// TIA Portal V20 export
VAR_GLOBAL   // PLC tag table "Robot_Efort"
   Mission_Command AT %QW524 : Int;   // Invio delle missioni a robot
   "X_Pick-Place_LOW" AT %QW526 : Int;
   "Y_Pick-Place_LOW" AT %QW530 : Int;
   "Z_Pick-Place_LOW" AT %QW534 : Int;
   "ZRot_Pick-Place_LOW" AT %QW538 : Int;
   "YRot_Pick-Place_LOW" AT %QW542 : Int;
   "XRot_Pick-Place_LOW" AT %QW546 : Int;
   Gripper_code AT %QW550 : Int;
   Gripper1_XDim_LOW AT %QW552 : Int;
   Gripper1_YDim_LOW AT %QW556 : Int;
   Gripper1_ZDim_LOW AT %QW560 : Int;
   Gripper1_ZRotDim_LOW AT %QW564 : Int;
   Gripper1_YRotDim_LOW AT %QW568 : Int;
   Gripper1_XRotDim_LOW AT %QW572 : Int;
   Gripper2_XDim_LOW AT %QW576 : Int;
   Gripper2_YDim_LOW AT %QW580 : Int;
   Gripper2_ZDim_LOW AT %QW584 : Int;
   Gripper2_ZRotDim_LOW AT %QW588 : Int;
   Gripper2_YRotDim_LOW AT %QW592 : Int;
   Gripper2_XRotDim_LOW AT %QW596 : Int;
   X_approach_LOW AT %QW600 : Int;
   Y_approach_LOW AT %QW604 : Int;
   Z_approach_LOW AT %QW608 : Int;
   ZRot_approach_LOW AT %QW612 : Int;
   YRot_approach_LOW AT %QW616 : Int;
   XRot_approach_LOW AT %QW620 : Int;
   ApproachType AT %QW624 : Int;   // 1 XX, 2 YY, 3 ZZ, 4 XZ, 5 ZX, 6 YZ, 7 ZY, 8 XY , 9 YX
   Unit_code AT %QW626 : Int;   // 1-4 warehouse, 11-14 Machines 1→4, 21-29 grippers positions 1→9 on shelf
   Object_Type AT %QW628 : Int;   // 1 Part, 2 vice, 3 pallet, 4 gripper
   Gripper_Side AT %QW632 : Int;   // 1 RAW, 2 fFINISHED
   cmd_Status_PalletLocked AT %Q503.0 : Bool;   // segnale di pallet bloccato
   cmd_Status_PalletUnlocked AT %Q503.1 : Bool;   // segnale di pallet sbloccato
   cmd_status_Vice_locked AT %Q503.2 : Bool;   // segnale di morsa chiusa
   cmd_status_Vice_unlocked AT %Q503.3 : Bool;   // segnale di morsa aperta
   cmd_status_DoorOpened AT %Q503.5 : Bool;   // segnale di porta aperta
   cmd_status_DoorClosed AT %Q503.4 : Bool;   // segnale di porta chiusa
   cmd_status_free_5 AT %Q503.7 : Bool;
   ACQ_PalletLockedReq AT %Q505.0 : Bool;   // Aknowledge di richiesta chiusura pallet
   ACQ_PalletUnlockedReq AT %Q505.1 : Bool;   // Aknowledge di richiesta apertura pallet
   ACQ_GripperLockedReq AT %Q505.2 : Bool;   // Aknowledge di richiesta chiusura Morsa
   ACQ_GripperUnlockedReq AT %Q505.3 : Bool;   // Aknowledge di richiesta apertura Morsa
   ACQ_DoorLockedReq AT %Q505.4 : Bool;   // Aknowledge di richiesta chiusura Porta
   Ok_Phase2 AT %Q502.3 : Bool;
   ACQ_DoorUnlockedReq AT %Q505.5 : Bool;   // Aknowledge di richiesta apertura Porta
   Ok_Phase2_MC AT %Q504.0 : Bool;
   Option_free_4 AT %Q507.1 : Bool;
   Option_free_5 AT %Q507.2 : Bool;
   Option_free_6 AT %Q507.3 : Bool;
   Option_free_7 AT %Q507.4 : Bool;
   Option_free_8 AT %Q507.5 : Bool;
   Option_free_9 AT %Q507.6 : Bool;
   Option_free_10 AT %Q507.7 : Bool;
   sys_RobotActSpeed AT %IW512 : Int;
   Command_Answer AT %IW532 : Int;   // 1 acquired, 2 in execution, 3 executed, 4 aborted 5 rifiutato, 6 interrupted
   sys_AxisSafePosition2 AT %I500.0 : Bool;   // MAINTENANCE POSITION
   sys_AxisSafePosition3 AT %I500.1 : Bool;   // PARKING POSITION
   sys_AxisSafePosition4 AT %I500.2 : Bool;   // HOME SU MACCHINA 1
   sys_LoadProgramComplete AT %I500.3 : Bool;
   sys_ServoConfirmState AT %I500.4 : Bool;   // Feedback comando di servo
   sys_reserveProgramAct AT %I500.5 : Bool;
   sys_ResetProgramState AT %I500.6 : Bool;   // FeedBack del comando di reset program
   sys_Heartbeat AT %I500.7 : Bool;
   sys_manual_T1 AT %I501.0 : Bool;   // Robot in manuale
   sys_Robot_Auto_Mode AT %I501.1 : Bool;   // Robot In Auto mode
   sys_manual_Full AT %I501.2 : Bool;   // Robot in manuale al 100% speed
   sys_servo_OK AT %I501.3 : Bool;   // Power ON Robot
   sys_Robot_AlarmState AT %I501.4 : Bool;   // Robot in allarme
   sys_Robot_EmergencyStopState AT %I501.5 : Bool;   // Emergenza Robot premuta
   sys_Robot_Run_State AT %I501.6 : Bool;   // Stao di Start (automatico + Power ON + Play)
   sys_AxisSafePosition1 AT %I501.7 : Bool;   // HOME POSITION
   sys_AxisSafePosition5 AT %I503.0 : Bool;   // HOME SU MACCHINA 2
   sys_AxisSafePosition6 AT %I503.1 : Bool;   // HOME SU MACCHINA 3
   sys_AxisSafePosition7 AT %I503.2 : Bool;   // HOME SU PALLET 1
   sys_AxisSafePosition8 AT %I503.3 : Bool;   // HOME SU PALLET 2
   sys_AlarmCode_1 AT %IW514 : Int;
   sys_AlarmCode_2 AT %IW516 : Int;
   sys_GetProgramNumber AT %IW518 : Int;
   sys_ReservedProgReset AT %IW520 : Int;
   sys_ReservedProgRun AT %IW522 : Int;
   sys_HeartBeat_counter AT %IW524 : Int;   // 13a Word
   GripperCodeMounted AT %IW534 : Int;   // Da verificare
   Alarmcode AT %IW530 : Int;
   Robot_IN_AREA AT %I503.5 : Bool;   // Robot fuori ingombro
   LOCAL_MODE AT %I502.4 : Bool;   // Da Verificare
   cmd_maintenance_free8 AT %Q630.0 : Bool;
   cmd_maintenance_free9 AT %Q630.1 : Bool;
   cmd_maintenance_free10 AT %Q630.2 : Bool;
   cmd_maintenance_free11 AT %Q630.3 : Bool;
   cmd_maintenance_OpenGripper1 AT %Q630.4 : Bool;
   cmd_maintenance_OpenGripper2 AT %Q630.5 : Bool;
   cmd_maintenance_GotoMaintenancePos AT %Q630.6 : Bool;
   cmd_maintenance_GotoHomePos AT %Q630.7 : Bool;
   cmd_maintenance_free AT %Q629.0 : Bool;
   cmd_maintenance_free_1 AT %Q629.1 : Bool;
   cmd_maintenance_free_2 AT %Q629.2 : Bool;
   cmd_maintenance_free_3 AT %Q629.3 : Bool;
   cmd_maintenance_free_4 AT %Q629.4 : Bool;
   cmd_maintenance_free_5 AT %Q629.5 : Bool;
   cmd_maintenance_free_6 AT %Q629.6 : Bool;
   cmd_maintenance_free_7 AT %Q629.7 : Bool;
   Sys_SetRobotspeed AT %QW512 : Int;   // set della velocità in percentuale (va refreshata ad ogni inizio ciclo e ad ogni allarme portandola a 0 e poi a quella impostata a pannello)
   Sys_setProgNumber AT %QW514 : Int;
   Sys_auxNumber AT %QW516 : Int;
   Sys_setAuxSpeed AT %QW518 : Int;
   Sys_reserveProgNum AT %QW520 : Int;
   Sys_mapPrgNum AT %QW522 : Int;
   Vice_ClawLength_mm AT %QW634 : Int;   // lunghezza chele morsa [mm]
   Part_Width_mm AT %QW636 : Int;   // larghezza pezzo [mm]
   X_Support_mm AT %QW638 : Int;   // quota di battuta [mm], 0 = spinta non configurata
   Part_Length_mm AT %QW640 : Int;
   Part_Height_mm AT %QW642 : Int;
   N_Cassetto AT %QW644 : Int;
   Z_Push_LOW AT %QW646 : Int;   // Z spinta, parola bassa (come X_Pick-Place_LOW)
   Z_Push_HIGH AT %QW648 : Int;   // Z spinta, parola alta (come X_Pick-Place_HIGH)
   spare_9 AT %QW650 : Int;
   spare_10 AT %QW652 : Int;
   spare_11 AT %QW654 : Int;
   spare_12 AT %QW656 : Int;
   spare_13 AT %QW658 : Int;
   spare_14 AT %QW660 : Int;
   spare_15 AT %QW662 : Int;
   spare_16 AT %QW664 : Int;
   spare_17 AT %QW666 : Int;
   sys_positionType AT %Q500.0 : Bool;
   sys_ServoEnable AT %Q500.4 : Bool;
   sys_ServoDisable AT %Q500.5 : Bool;   // Disabilita i motori (va a 0 quando vedo servostate a 0)
   sys_loadMapPrg AT %Q500.7 : Bool;
   sys_servoOn AT %Q501.0 : Bool;   // Abilitazione servo robot (va a 0 quando vedo servo state a 1)
   sys_startProg AT %Q501.1 : Bool;   // Abilitaizone per la partenza (va a 0 quando vedo lo run state a 1)
   sys_pauseProgram AT %Q501.2 : Bool;   // Stop di congelamento in ciclo (il robot si ferma ma è pronto a ripartire esattamente da dove era per concludere il ciclo) (segnale da abbassare quando vedo runstate che va a 0)
   sys_resetAlarm AT %Q501.3 : Bool;   // Reset degli allarmi (quando vedo il systemalamstate che va a 0 il segnale va a 0)
   sys_loadProgram AT %Q501.4 : Bool;   // NON UTILIZZATO
   sys_resetProgram AT %Q501.5 : Bool;   // PP to main del programma (va a 0 quando vedo on resetprogramstate)
   sys_plcAlarm AT %Q501.6 : Bool;   // Segnale d'allarme da PLC
   sys_remoteServoConfirm AT %Q501.7 : Bool;   // Segnale di remote servo (va a 0 quando servoconfirmstate va a 1)
   cmd_ACK_Blowing AT %Q502.0 : Bool;   // Acknowladge della richiesta di soffio
   cmd_ACK_Washing AT %Q502.1 : Bool;   // Acknowladge della richiesta di lavaggio
   px_tray_in_position AT %Q502.4 : Bool;   // Sensore di cassetto estratto
   cmd_status_free_3 AT %Q502.5 : Bool;
   cmd_status_Gripper_1_Ready AT %Q502.6 : Bool;   // Presenza delle ganasce nalla posizione 1 della pinza
   cmd_status_Gripper_2_Ready AT %Q502.7 : Bool;   // Presenza delle ganasce nalla posizione 2 della pinza
   Gripper_mounted AT %I502.0 : Bool;   // Pinza montata
   Gripper1_Closed AT %I502.1 : Bool;   // Pinza 1 chiusa
   Gripper2_Closed AT %I502.2 : Bool;   // Pinza 2 chiusa
   Robot_cmd_free2 AT %I504.1 : Bool;
   Robot_PushDepositoFatto_MC AT %I504.2 : Bool;
   Robot_PushInPos_MC AT %I504.3 : Bool;
   Robot_cmd_free5 AT %I504.4 : Bool;
   Robot_cmd_free6 AT %I504.5 : Bool;
   Robot_cmd_free7 AT %I504.6 : Bool;
   Robot_cmd_free8 AT %I504.7 : Bool;
   Robot_cmd_LockPallet AT %I505.0 : Bool;   // Richiesta di sblocco pallet da robot
   Robot_cmd_UnlockPallet AT %I505.1 : Bool;   // Richiesta di blocco pallet da robot
   Robot_cmd_LockPart AT %I505.2 : Bool;   // Richiesta di chiusura morsa da robot
   Robot_cmd_UnlockPart AT %I505.3 : Bool;   // richiesta di apertura morsa da robot
   Robot_cmd_OpenDoor AT %I505.4 : Bool;   // richiesta di apertura porta da robot
   Robot_cmd_CloseDoor AT %I505.5 : Bool;   // richiesta di chiusura porta da robot
   Robot_cmd_BLOW AT %I505.6 : Bool;   // richiesta di soffiaggio da robot
   Robot_cmd_WASHING AT %I505.7 : Bool;   // richiesta di lavaggio da robot
   newQuotaReady AT %I511.7 : Bool;   // Da verificare
   RobotPosition_J1X AT %ID540 : Real;   // Quota asse J1
   RobotPosition_J2Y AT %ID544 : Real;   // Quota asse J2
   RobotPosition_J3Z AT %ID548 : Real;   // Quota asse J3
   RobotPosition_J4A AT %ID552 : Real;   // Quota asse J4
   RobotPosition_J5B AT %ID556 : Real;   // Quota asse J5
   RobotPosition_J6C AT %ID560 : Real;   // Quota asse J6
   sys_connfirmReservProgram AT %Q500.1 : Bool;
   sys_cancelReserveProgram AT %Q500.2 : Bool;
   sys_reservProgramOnOff AT %Q500.3 : Bool;
   "Y_Pick-Place_HIGH" AT %QW532 : Int;
   "X_Pick-Place_HIGH" AT %QW528 : Int;
   "Z_Pick-Place_HIGH" AT %QW536 : Int;
   "ZRot_Pick-Place_HIGH" AT %QW540 : Int;
   "YRot_Pick-Place_HIGH" AT %QW544 : Int;
   "XRot_Pick-Place_HIGH" AT %QW548 : Int;
   Gripper1_XDim_HIGH AT %QW554 : Int;
   Gripper1_YDim_HIGH AT %QW558 : Int;
   Gripper1_ZDim_HIGH AT %QW562 : Int;
   Gripper1_ZRotDim_HIGH AT %QW566 : Int;
   Gripper1_YRotDim_HIGH AT %QW570 : Int;
   Gripper1_XRotDim_HIGH AT %QW574 : Int;
   Gripper2_XDim_HIGH AT %QW578 : Int;
   Gripper2_YDim_HIGH AT %QW582 : Int;
   Gripper2_ZDim_HIGH AT %QW586 : Int;
   Gripper2_ZRotDim_HIGH AT %QW590 : Int;
   Gripper2_YRotDim_HIGH AT %QW594 : Int;
   Gripper2_XRotDim_HIGH AT %QW598 : Int;
   X_approach_HIGH AT %QW602 : Int;
   Y_approach_HIGH AT %QW606 : Int;
   Z_approach_HIGH AT %QW610 : Int;
   ZRot_approach_HIGH AT %QW614 : Int;
   YRot_approach_HIGH AT %QW618 : Int;
   XRot_approach_HIGH AT %QW622 : Int;
   Area_output_1 AT %I503.4 : Bool;   // Area di lavoro del robot (lavora sempre a 1 e se il robot è spento va a 0)
   Robot_SwapPhase2Req AT %I502.3 : Bool;   // Bit di passaggio a fase 2 della missione
   Area_output_2 AT %I502.5 : Bool;   // Fori ingombro dalla macchina
   Area_output_3 AT %I503.6 : Bool;   // Area libera da configurare
   Area_output_4 AT %I503.7 : Bool;   // Area libera da configurare
   Robot_Phase2Req_MC AT %I504.0 : Bool;
   Q_PushEnable_MC AT %Q504.1 : Bool;
   Ok_PushSpinta_MC AT %Q504.2 : Bool;
   Ok_PushArrivo_MC AT %Q504.3 : Bool;
   cmd_MC_auto AT %Q503.6 : Bool;   // segnale di macchina in automatico
   Home_Speed AT %IW526 : Int;   // Velocità da robot durante il ritorno in home
END_VAR
